// TIA Portal V19 export
FUNCTION_BLOCK "TYPIC_C301_SF_VEN_CLUST"   // FB7, FBD
TITLE = TYPIC_C301_SF_VEN_CLUST: Ventilatiecluster verkeerskoker
{ S7_Optimized_Access := 'TRUE' }
AUTHOR : OCOTECH
FAMILY : Typical
NAME : C301.802
// Logisch Object Besturing: C301.802
// 
// Het doel van de SF ventilatiecluster is het aansturen van een cluster van ventilatoren op basis van sturingen ontvangen van de basisfunctie “ventilatie”, bedieningen op IRIS SCADA en de status van de aangestuurde ventilatoren
// stored: MemoryReserve 10, SetENOAutomatically false
   VAR_INPUT
      CFG_NUM { ExternalAccessible := 'False'; ExternalVisible := 'False'; ExternalWritable := 'False'} : USInt;   // Nummer van de cluster binnen ventilatiezone 0 = ingangscluster
      CFG_TYD_ONHD1 { ExternalAccessible := 'False'; ExternalVisible := 'False'; ExternalWritable := 'False'} : USInt;   // Tijdsduur aansturing ventilator bij automatische onderhoudstesten
      CFG_TYD_ONHD2 { ExternalAccessible := 'False'; ExternalVisible := 'False'; ExternalWritable := 'False'} : USInt;   // Tijdsduur intervaltijd bij automatische onderhoudstesten
      STU_CMD_AUT { ExternalAccessible := 'False'; ExternalVisible := 'False'; ExternalWritable := 'False'} : USInt;   // Groepscommando: schakel in automatisch
      STU_ALG_LCK_SIG { ExternalAccessible := 'False'; ExternalVisible := 'False'; ExternalWritable := 'False'} : USInt;   // Onderdruk alarmen
      STU_ENE_VGV_AAN { ExternalAccessible := 'False'; ExternalVisible := 'False'; ExternalWritable := 'False'} : USInt;   // Vrijgeven of verhinderen bijschakelen energieverbruikers (verlichting / ventilatie)
      STU_ENE_MAX_AAN { ExternalAccessible := 'False'; ExternalVisible := 'False'; ExternalWritable := 'False'} : USInt;   // Maximaal toegelaten ventilatiestand
   END_VAR
   VAR_OUTPUT
      VAR_CLUST { ExternalAccessible := 'False'; ExternalVisible := 'False'; ExternalWritable := 'False'} : "C301_VAR_CLUST_TYPIC";   // Struct met alle variabelen van de cluster (info naar de bovenliggende basisfunctie)
      STU_VEN1 { ExternalAccessible := 'False'; ExternalVisible := 'False'; ExternalWritable := 'False'} : "C301_STU_VEN_TYPIC";   // sturing naar ventilator 1
      STU_VEN2 { ExternalAccessible := 'False'; ExternalVisible := 'False'; ExternalWritable := 'False'} : "C301_STU_VEN_TYPIC";   // sturing naar ventilator 2
      STU_VEN3 { ExternalAccessible := 'False'; ExternalVisible := 'False'; ExternalWritable := 'False'} : "C301_STU_VEN_TYPIC";   // sturing naar ventilator 3
      STU_VEN4 { ExternalAccessible := 'False'; ExternalVisible := 'False'; ExternalWritable := 'False'} : "C301_STU_VEN_TYPIC";   // sturing naar ventilator 4
      STU_VEN5 { ExternalAccessible := 'False'; ExternalVisible := 'False'; ExternalWritable := 'False'} : "C301_STU_VEN_TYPIC";   // sturing naar ventilator 5
      STU_VEN6 { ExternalAccessible := 'False'; ExternalVisible := 'False'; ExternalWritable := 'False'} : "C301_STU_VEN_TYPIC";   // sturing naar ventilator 6
      STU_VEN7 { ExternalAccessible := 'False'; ExternalVisible := 'False'; ExternalWritable := 'False'} : "C301_STU_VEN_TYPIC";   // sturing naar ventilator 7
      STU_VEN8 { ExternalAccessible := 'False'; ExternalVisible := 'False'; ExternalWritable := 'False'} : "C301_STU_VEN_TYPIC";   // sturing naar ventilator 8
   END_VAR
   VAR_IN_OUT
      CFG_CAPA_DIR1 : Array[1..8] of USInt;   // Omzetting ventilatiestand naar aantal ventilatoren, per cluster (zie verder), rijrichting
      CFG_CAPA_DIR2 : Array[1..8] of USInt;   // Omzetting ventilatiestand naar aantal ventilatoren, per cluster (zie verder), tegenrijrichting
      VAR_VEN : Array[*] of "C301_VAR_VEN_TYPIC";   // Array met alle ventilatoren, met alle variabelen van de ventilator
      STU_CLUST : "C301_STU_CLUST_TYPIC";   // Struct met alle sturingen vanuit de basisfunctie naar de cluster
   END_VAR
   VAR
      BED : Struct   // Bedieningen
         ALG : Struct   // Gewenste stand
            X : "UDT_BED_ALG";
            KNOP { S7_SetPoint := 'True'} : Array[0..2] of "UDT_BED_KNOP";
         END_STRUCT;
         BST : Struct   // Bestuurbaarheid
            X : "UDT_BED_ALG";
            KNOP { S7_SetPoint := 'True'} : Array[0..1] of "UDT_BED_KNOP";
         END_STRUCT;
      END_STRUCT;
      BED_ALG { ExternalWritable := 'False'} : "TYPIC_HF_BED_ALG_KNOP";   // Gewenste stand
      BED_BST { ExternalWritable := 'False'} : "TYPIC_HF_BED_ALG_KNOP";   // Bestuurbaarheid
      VAR { ExternalWritable := 'False'} : Struct   // Variabelen
         CAPA : USInt;   // Gewenste capaciteitsinstelling
         NIV_SWA { ExternalAccessible := 'False'; ExternalVisible := 'False'} : USInt;   // Gewenst aantal aangeschakelde ventilatoren
         ONHD_VEN { ExternalAccessible := 'False'; ExternalVisible := 'False'} : USInt;   // Nummer ventilator bezig met onderhoudstest
         STU { ExternalAccessible := 'False'; ExternalVisible := 'False'} : USInt;   // Array met de sturingen naar iedere ventilator
         CAPA_OK { ExternalAccessible := 'False'; ExternalVisible := 'False'} : USInt;   // Aantal bestuurbare ventilatoren in de cluster
         NIV_AAN_BWA : USInt;   // Aantal aangeschakelde ventilatoren in de gewenste ventilatierichting
         DIR : USInt;   // Richting van de cluster
         BMO : USInt;   // Bedieningsmode
         ONHD_STS : USInt;   // Status automatische onderhoudstesten
         PWR { ExternalAccessible := 'False'; ExternalVisible := 'False'} : Real;   // Actueel vermogen van de ventilatiecluster
      END_STRUCT;
   END_VAR
   // // BED.ALG.KNOP[0] : Auto
   // // BED.ALG.KNOP[1] : 0 (Uit)
   // // BED.ALG.KNOP[2] : 8
   // // BED.BST.KNOP[0] : InDienst
   // // BED.BST.KNOP[1] : UitDienst
BEGIN

REGION Network 1: START
END_REGION

REGION Network 2: +++ Bedieningen +++
   // Vrijgave en verwerking van de bedieningen (centrale en lokale bediening). De bedienwaardes worden daarna in de verdere deelfunctionaliteiten gebruikt.
END_REGION

REGION Network 3: Knoppen BED_ALG(Gewenste stand)
   // Waardes en vrijge van de knoppen BED_ALG
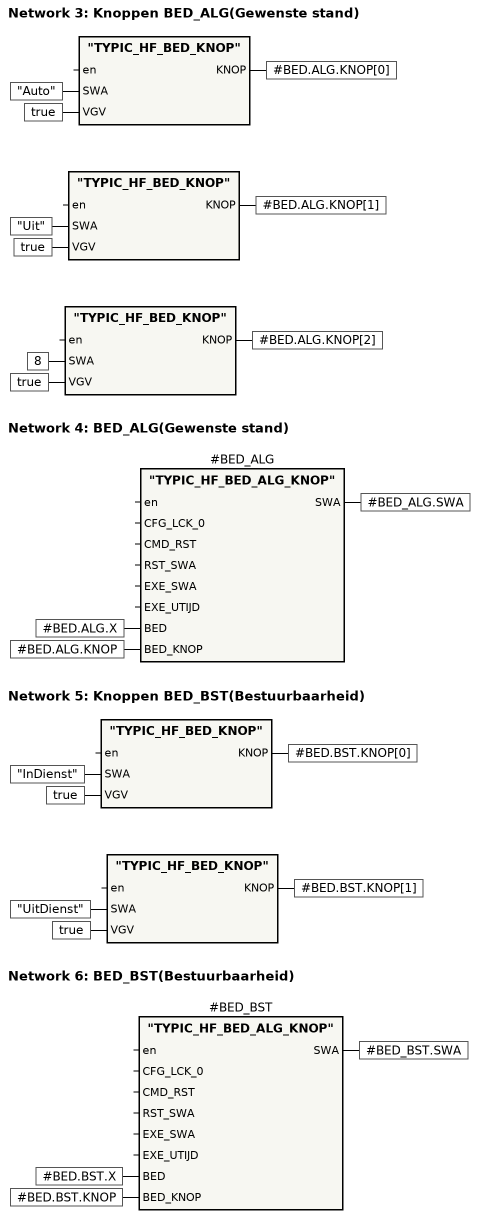
   "TYPIC_HF_BED_KNOP"(SWA := "Auto", VGV := true, KNOP => #BED.ALG.KNOP[0]);
   "TYPIC_HF_BED_KNOP"(SWA := "Uit", VGV := true, KNOP => #BED.ALG.KNOP[1]);
   "TYPIC_HF_BED_KNOP"(SWA := 8, VGV := true, KNOP => #BED.ALG.KNOP[2]);
END_REGION

REGION Network 4: BED_ALG(Gewenste stand)
   // Verwerking BED_ALG
   #BED_ALG(BED := #BED.ALG.X, BED_KNOP := #BED.ALG.KNOP, SWA => #BED_ALG.SWA);   // "TYPIC_HF_BED_ALG_KNOP"
END_REGION

REGION Network 5: Knoppen BED_BST(Bestuurbaarheid)
   // Waardes en vrijge van de knoppen BED_BST
   "TYPIC_HF_BED_KNOP"(SWA := "InDienst", VGV := true, KNOP => #BED.BST.KNOP[0]);
   "TYPIC_HF_BED_KNOP"(SWA := "UitDienst", VGV := true, KNOP => #BED.BST.KNOP[1]);
END_REGION

REGION Network 6: BED_BST(Bestuurbaarheid)
   // Verwerking BED_BST
   #BED_BST(BED := #BED.BST.X, BED_KNOP := #BED.BST.KNOP, SWA => #BED_BST.SWA);   // "TYPIC_HF_BED_ALG_KNOP"
END_REGION

REGION Network 7: +++ Bepalen bedieningsmode en gewenste capaciteitsinstelling +++
   // Bedieningsmode (Auto / Manueel ) bepalen en gewenste stand (0..8) bepalen
END_REGION

REGION Network 8: +++ Bepalen werkelijke ventilatierichting +++
   // Bepalen van de werkelijke ventilatierichting (Rijrichting / Tegenrij / Onbepaald) aan de hand van de ventilatierichtingen van de ventilatieclusters.
END_REGION

REGION Network 9: +++ Bepalen gewenst aantal ventilatoren +++
   // Bepalen van het gewenst aantal ingeschakelde ventilatoren.
END_REGION

REGION Network 10: +++ Bepalen aansturing ventilatoren +++
   // Sturing van iedere individuele ventilator bepalen op basis van de werkingsmode en bestuurbaarheid van de ventilator en de gewenste draairichting van de cluster
END_REGION

REGION Network 11: +++ Berekeningen +++
   // Verscheidene berekeningen die nodig zijn voor de functionele werking of info voor weergave via de centrale en lokale bediening, zoals het  aantal bestuurbare ventilatoren, aantal ventilatoren aangestuurd in draairichting, actueel vermogen van de ventilatiecluster
END_REGION

REGION Network 12: +++ Bij- of afschakelen ventilator +++
   // Bijschakelen van de ventilator met het minst aantal draaiuren als aantal aangeschakelde ventilatoren lager dan het gewenst aantal. Afschakelen van de ventilator met meest aantal draaiuren als het aantal aangeschakelde ventilatoren hoger is dan het gewenst aantal.
END_REGION

REGION Network 13: +++ Automatische onderhoudstesten +++
   // Functionaliteit waarbij iedere ventilator een voor een aangestuurd wordt ter controle van de goede werking van iedere ventilator.
END_REGION

REGION Network 14: +++ Sturingen +++
   // Uitgeven van sturingen naar de ventilatoren.
END_REGION

REGION Network 15 (SCL): EINDE
   // Variabelen van intern scada rakvlak naar outputs copieren
   #VAR_CLUST.CAPA_OK := #VAR.CAPA_OK;
   #VAR_CLUST.NIV_AAN_BWA := #VAR.NIV_AAN_BWA;
   #VAR_CLUST.DIR := #VAR.DIR;
   #VAR_CLUST.BMO := #VAR.BMO;
   #VAR_CLUST.ONHD_STS := #VAR.ONHD_STS;
   #VAR_CLUST.PWR := #VAR.PWR;
END_REGION
END_FUNCTION_BLOCK
